PROGRAM MAIN
VAR
	rRoundedValue 	: ARRAY[1..6] OF REAL;
	rRawValue		: ARRAY[1..6] OF REAL := [1.111,2.222,3.666,4.888,5.555,6.159];
END_VAR

rRoundedValue := F_ROUND_REAL(rRawValue, 1);
GVL.rRoundedValue := F_ROUND_REAL_GLOBAL(1);

END_PROGRAM

(* stored: Version 1.1.0.1, ProductVersion 3.1.4024.12
   POU MAIN: Id {bd6446df-a555-4a9a-9801-8a139cc9f785}, SpecialFunc None *)
